// TIA Portal V20 export
DATA_BLOCK "ET200SP_203"   // DB272
// stored: MemoryReserve 100
   VAR
      "SP203.00 Main OP: mode select, Auto" : Bool;
      "SP203.01 Main OP: home (GREEN)" : Bool;
      "SP203.02 Main OP: safety reset (BLUE)" : Bool;
      "SP203.03 Main OP: SCS mode select, Auto" : Bool;
      "SP203.04 Main OP: mode select, Manual" : Bool;
      "SP203.05 Main OP: enable" : Bool;
      "SP203.06 Main OP: SCS mode select, Setup" : Bool;
      "SP203.07 Main OP: SCS mode select, Disable" : Bool;
   END_VAR
BEGIN
END_DATA_BLOCK
